// TIA Portal V20 export
DATA_BLOCK "DB_DataLog"   // DB12
{ S7_Optimized_Access := 'TRUE' }
// stored: MemoryReserve 100
   VAR
      Create_DataLog : Bool;
      Open_DataLog : Bool;
      Write_DataLog : Bool;
      Close_DataLog : Bool;
      Clean_DataLog : Bool;
      Delete_DataLog : Bool;
      ID_DataLog : DWord;
      Name_DataLog : String := 'Teste Funcional';
      Header_DataLog : String := 'Bebedoro,Numero de Serie,Painel,Tensao Eletrica [V],Corrente Eletrica [mA],Resultado Teste Corrente,Resultado Teste Visual,Resultado Teste Funcional';
   END_VAR
BEGIN
END_DATA_BLOCK
